FUNCTION_BLOCK FB_SVs_Input
VAR_INPUT
	IN_Zustand_Stellungrueckmeldung0 : BOOL;
	IN_Zustand_Stellungrueckmeldung1 : BOOL;

END_VAR
VAR_OUTPUT
	Zustand_Stellungrueckmeldung0 : BOOL;
	Zustand_Stellungrueckmeldung1 : BOOL;

END_VAR
VAR
END_VAR

Zustand_Stellungrueckmeldung0 := IN_Zustand_Stellungrueckmeldung0;
Zustand_Stellungrueckmeldung1 := IN_Zustand_Stellungrueckmeldung1;

END_FUNCTION_BLOCK

(* stored: Version 1.1.0.1, ProductVersion 3.1.4024.9
   POU FB_SVs_Input: Id {a42ea13d-a8f5-4e1d-b883-1c08f29984df}, SpecialFunc None *)
